ABB RobotStudio station: CV_1_homework.rspag

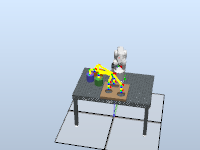
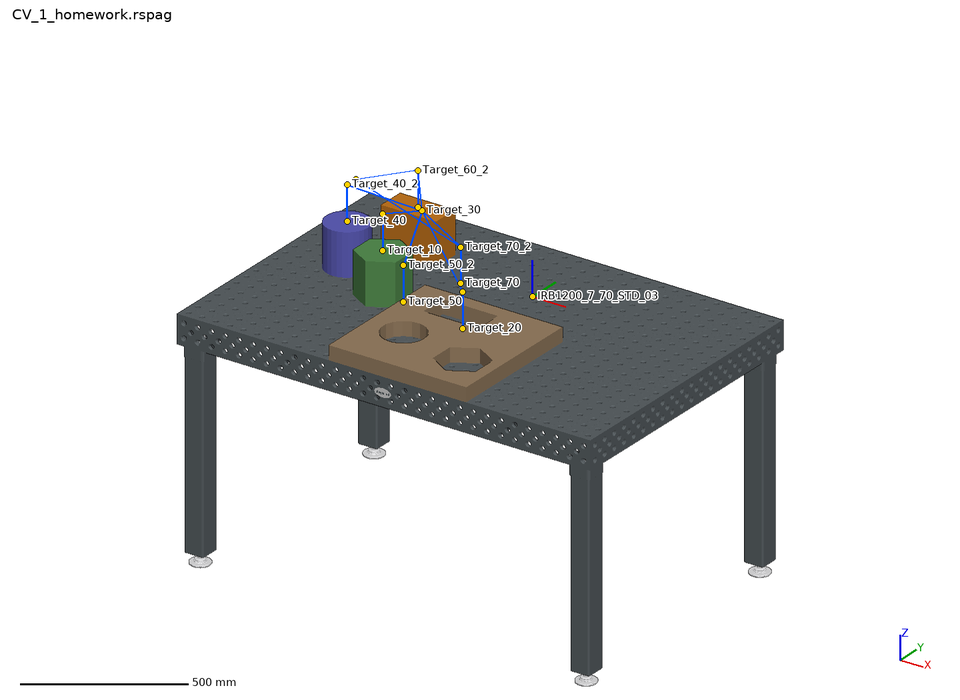
[picture v1: parts stored in the station drawn from their meshes, with robot base, taught points and paths (robot models come from the ABB library and are not in the file)]
--- station ---
Station Solution_1_Tutorial (saved by RobotStudio 21.4.9700.0)
Controller Controller2, task T_ROB1: task frame (RAPID world) sits at (50, 200, 830) mm, rotated rx 0 ry 0 rz -90 deg in the station
Controller Controller2
  mechanical unit ROB_1: IRB1200_7_70_STD_03, 6 joints, base frame (0, 0, 0) mm
Layout (positions relative to the parent item):
  - table [part] at (-200, -500, 830) mm, size 500 x 500 x 50 mm
  - object_1 [part] at (-600, -150, 830) mm, size 200 x 100 x 150 mm
  - object_2 [part] at (-650, -150, 830) mm, size 149.5 x 149.7 x 150 mm
  - object_3 [part] at (-700, -200, 830) mm, size 155.5 x 179.5 x 150 mm
  - siegmund_1500_1000 [part], size 1500 x 1010.3 x 830 mm
  - object_11 [part] at (-200, -500, 830) mm, size 200 x 100 x 150 mm
  - object_22 [part] at (-200, -500, 830) mm, size 149.5 x 149.7 x 150 mm
  - object_33 [part] at (-200, -500, 830) mm, size 155.5 x 179.5 x 150 mm
  - IRB1200_7_70_STD_03 [mechanism, from Robots\IRB1200_7_70_STD_03.rslib] at (50, 200, 830) mm, rotated rx 0 ry 0 rz -90 deg; joint values [0.2295, 0.4775, -0.4298, -0.6469, 1.6733, 1.7819] (rad or m)
  - MyTool [mechanism, from Training Objects\myTool.rslib] at (116.33, -300, 1500.53) mm, rotated rx -180 ry 38 rz 0 deg
  - Positioner [smart component, from Components\Positioner.rslib]
      properties: Object=object_1; Position=[-0.6 -0.15 0.83]; Orientation=[0 0 0]; Reference=Global; ReferenceObject=(none)
  - Positioner_2 [smart component, from Components\Positioner.rslib]
      properties: Object=object_2; Position=[-0.65 -0.15 0.83]; Orientation=[0 0 0]; Reference=Global; ReferenceObject=(none)
  - Positioner_3 [smart component, from Components\Positioner.rslib]
      properties: Object=object_3; Position=[-0.7 -0.2 0.83]; Orientation=[0 0 0]; Reference=Global; ReferenceObject=(none)
  - Attacher [smart component, from Components\Attacher.rslib]
      properties: Parent=MyTool; Flange=0; Child=object_3; Mount=false; Offset=[0 0 0]; Orientation=[0 0 0]
  - Detacher [smart component, from Components\Detacher.rslib]
      properties: Child=object_3; KeepPosition=true
  - Attacher_2 [smart component, from Components\Attacher.rslib]
      properties: Parent=MyTool; Flange=0; Child=object_2; Mount=false; Offset=[0 0 0]; Orientation=[0 0 0]
  - Detacher_2 [smart component, from Components\Detacher.rslib]
      properties: Child=object_2; KeepPosition=true
  - Attacher_3 [smart component, from Components\Attacher.rslib]
      properties: Parent=MyTool; Flange=0; Child=object_1; Mount=false; Offset=[0 0 0]; Orientation=[0 0 0]
  - Detacher_3 [smart component, from Components\Detacher.rslib]
      properties: Child=object_1; KeepPosition=true
Attachment: MyTool is attached to IRB1200_7_70_STD_03 / Link6
Station signals: DI di_pos_obj1, DI di_pos_obj2, DI di_pos_obj3
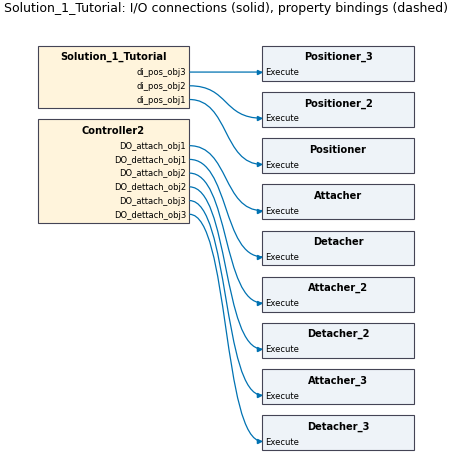
Station logic (signal -> signal, property => property):
  Solution_1_Tutorial.di_pos_obj3 -> Positioner_3.Execute
  Solution_1_Tutorial.di_pos_obj2 -> Positioner_2.Execute
  Solution_1_Tutorial.di_pos_obj1 -> Positioner.Execute
  Controller2.DO_attach_obj1 -> Attacher.Execute
  Controller2.DO_dettach_obj1 -> Detacher.Execute
  Controller2.DO_attach_obj2 -> Attacher_2.Execute
  Controller2.DO_dettach_obj2 -> Detacher_2.Execute
  Controller2.DO_attach_obj3 -> Attacher_3.Execute
  Controller2.DO_dettach_obj3 -> Detacher_3.Execute
Targets, tools, work objects and paths stored in the station and not in the controller backup, written as RAPID:
! task T_ROB1
MODULE CalibData
  PERS tooldata Servo:=[TRUE,[[0,0,84],[1,0,0,0]],[0.226,[8.9,12.3,48.7],[1,0,0,0],0.00021,0.00024,0.00009]];
  PERS tooldata VaccumOne:=[TRUE,[[63.5,18.5,37.5],[0.707106781,0,0.707106781,0]],[0.226,[8.9,12.3,48.7],[1,0,0,0],0.00021,0.00024,0.00009]];
ENDMODULE


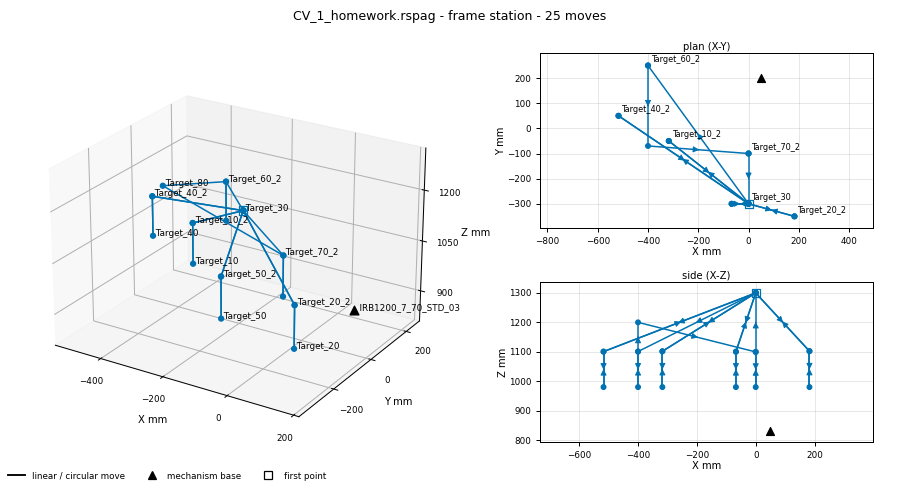
[picture p0: tool path of CV_1_homework.rspag in frame station, 25 of 25 moves have a stored position in this frame; points joined in program order, loops and branches not executed]
--- Backups/Controller2/RAPID/TASK1/PROGMOD/CalibData.mod ---
MODULE CalibData
    PERS tooldata MyTool:=[TRUE,[[31.792631019,0,229.638935148],[0.945518576,0,0.325568154,0]],[1,[0,0,1],[1,0,0,0],0,0,0]];
ENDMODULE

--- Backups/Controller2/RAPID/TASK1/PROGMOD/Module1.mod ---
MODULE Module1

        CONST robtarget Target_30:=[[500,-50,470],[0,0.707106781,0.707106781,0],[0,0,0,0],[9E+09,9E+09,9E+09,9E+09,9E+09,9E+09]];
    CONST robtarget Target_10_2:=[[250,-367.298,271.606391864],[0,0.707106781,0.707106781,0],[-1,-1,1,0],[9E+09,9E+09,9E+09,9E+09,9E+09,9E+09]];
    CONST robtarget Target_10:=[[250,-367.298,150],[0,0.707106781,0.707106781,0],[-1,-2,1,0],[9E+09,9E+09,9E+09,9E+09,9E+09,9E+09]];
    CONST robtarget Target_20_2:=[[550,132.702,272.182572429],[0,0.707106781,0.707106781,0],[0,0,0,0],[9E+09,9E+09,9E+09,9E+09,9E+09,9E+09]];
    CONST robtarget Target_20:=[[550,132.702,150],[0,0.707106781,0.707106781,0],[0,0,0,0],[9E+09,9E+09,9E+09,9E+09,9E+09,9E+09]];
    CONST robtarget Target_40_2:=[[150,-567.298,270.556474703],[0,0.707106781,0.707106781,0],[-1,-1,0,0],[9E+09,9E+09,9E+09,9E+09,9E+09,9E+09]];
    CONST robtarget Target_40:=[[150,-567.298,150],[0,0.707106781,0.707106781,0],[-1,-2,1,0],[9E+09,9E+09,9E+09,9E+09,9E+09,9E+09]];
    CONST robtarget Target_50_2:=[[500,-117.298,270.367811283],[0,0.707106781,0.707106781,0],[0,-1,1,0],[9E+09,9E+09,9E+09,9E+09,9E+09,9E+09]];
    CONST robtarget Target_50:=[[500,-117.298,150],[0,0.707106781,0.707106781,0],[0,-1,1,0],[9E+09,9E+09,9E+09,9E+09,9E+09,9E+09]];
    CONST robtarget Target_60_2:=[[-50,-450,270.839115212],[0,0.707106781,0.707106781,0],[-2,0,-1,0],[9E+09,9E+09,9E+09,9E+09,9E+09,9E+09]];
    CONST robtarget Target_60:=[[-50,-450,150],[0,0.707106781,0.707106781,0],[-2,1,-2,0],[9E+09,9E+09,9E+09,9E+09,9E+09,9E+09]];
    CONST robtarget Target_80:=[[270,-450,370],[0,0.707106781,0.707106781,0],[-1,-1,0,0],[9E+09,9E+09,9E+09,9E+09,9E+09,9E+09]];
    CONST robtarget Target_70_2:=[[300,-50,269.482150799],[0,0.707106781,0.707106781,0],[0,-1,1,0],[9E+09,9E+09,9E+09,9E+09,9E+09,9E+09]];
    CONST robtarget Target_70:=[[300,-50,150],[0,0.707106781,0.707106781,0],[0,-1,1,0],[9E+09,9E+09,9E+09,9E+09,9E+09,9E+09]];
PROC main()
    Path_10;
    ENDPROC
    PROC Path_10()
        MoveL Target_30,v200,fine,MyTool\WObj:=wobj0;

        !PICK1
        MoveL Target_10_2,v200,fine,MyTool\WObj:=wobj0;
        MoveL Target_10,v200,fine,MyTool\WObj:=wobj0;
        WaitTime 0.1;
        PulseDO DO_attach_obj1;
        WaitTime 0.1;
        MoveL Target_10_2,v200,fine,MyTool\WObj:=wobj0;
        MoveL Target_30,v200,fine,MyTool\WObj:=wobj0;

        !PLACE1
        MoveL Target_20_2,v200,fine,MyTool\WObj:=wobj0;
        MoveL Target_20,v200,fine,MyTool\WObj:=wobj0;
        WaitTime 0.1;
        PulseDO DO_dettach_obj1;
        WaitTime 0.1;
        MoveL Target_20_2,v200,fine,MyTool\WObj:=wobj0;
        MoveL Target_30,v200,fine,MyTool\WObj:=wobj0;

        !PICK2
        MoveL Target_40_2,v200,fine,MyTool\WObj:=wobj0;
        MoveL Target_40,v200,fine,MyTool\WObj:=wobj0;
        WaitTime 0.1;
        PulseDO DO_attach_obj2;
        WaitTime 0.1;
        MoveL Target_40_2,v200,fine,MyTool\WObj:=wobj0;
        MoveL Target_30,v200,fine,MyTool\WObj:=wobj0;

        !PLACE2
        MoveL Target_50_2,v200,fine,MyTool\WObj:=wobj0;
        MoveL Target_50,v200,fine,MyTool\WObj:=wobj0;
        WaitTime 0.1;
        PulseDO DO_dettach_obj2;
        WaitTime 0.1;
        MoveL Target_50_2,v200,fine,MyTool\WObj:=wobj0;
        MoveL Target_30,v200,fine,MyTool\WObj:=wobj0;

        !PICK3
        MoveL Target_60_2,v200,fine,MyTool\WObj:=wobj0;
        MoveL Target_60,v200,fine,MyTool\WObj:=wobj0;
        WaitTime 0.1;
        PulseDO DO_attach_obj3;
        WaitTime 0.1;
        MoveL Target_60_2,v200,fine,MyTool\WObj:=wobj0;
        MoveL Target_80,v200,fine,MyTool\WObj:=wobj0;

        !PLACE3
        MoveL Target_70_2,v200,fine,MyTool\WObj:=wobj0;
        MoveL Target_70,v200,fine,MyTool\WObj:=wobj0;
        WaitTime 0.1;
        PulseDO DO_dettach_obj3;
        WaitTime 0.1;
        MoveL Target_70_2,v200,fine,MyTool\WObj:=wobj0;
        MoveL Target_30,v200,fine,MyTool\WObj:=wobj0;
    ENDPROC
ENDMODULE

--- Backups/Controller2/SYSPAR/EIO.cfg ---
EIO:CFG_1.0:6:1::
#
EIO_SIGNAL:

      -Name "DO_attach_obj1" -SignalType "DO"

      -Name "DO_attach_obj2" -SignalType "DO"

      -Name "DO_attach_obj3" -SignalType "DO"

      -Name "DO_dettach_obj1" -SignalType "DO"

      -Name "DO_dettach_obj2" -SignalType "DO"

      -Name "DO_dettach_obj3" -SignalType "DO"
